// TIA Portal project "babu_washingMachineHMI" (V15)

(* hardware
DEVICE "S7-1200 station_1"  S7-1200 Station
   slot 0: "Rack_0"  S7-1200 Rack  Rack  V1.0
   slot 1: "PLC_1"  CPU 1212C DC/DC/DC  6ES7 212-1AE40-0XB0  V4.2
DEVICE "HMI_1"  KTP400 Basic PN
   slot 0: "HMI_1"  KTP400 Basic PN  6AV2 123-2DB03-0AX0  15.0.0.0
   slot 1: "HMI_RT_1"  KTP400 Basic PN  6AV2 123-2DB03-0AX0  15.0.0.0
   slot 5: "HMI_1.IE_CP_1"  PROFINET Interface  15.0.0.0
      slot 1: "PROFINET Interface_1"  PROFINET Interface
         slot 1: "Port_1"  Port
*)

// ===== PLC "PLC_1"  CPU 1212C DC/DC/DC =====

VAR_GLOBAL   // PLC tag table "Default tag table"
   "PUSH BUTTON ON" AT %M0.0 : Bool;
   "PUSH BUTTON ON MEM" AT %M0.1 : Bool;
   "PUSH BUTTON STOP" AT %M0.2 : Bool;
   "PUSH BUTTON STOP MEM" AT %M0.3 : Bool;
   "WATER AVAILABLE" AT %M0.4 : Bool;
   "WATER AVAILABLE MEM" AT %M0.5 : Bool;
   "DOOR CLOSED" AT %M0.6 : Bool;
   "DOOR CLOSED MEM" AT %M0.7 : Bool;
   "CLOTHS AVAILABLE MEM" AT %M1.0 : Bool;
   "CLOTHS AVAILABLE" AT %M1.1 : Bool;
   "CLEANING SOLUTION AVAILABLE" AT %M1.2 : Bool;
   "CLEANING SOLUTION AVAILABLE MEM" AT %M1.3 : Bool;
   "ALL OK TO START" AT %M1.4 : Bool;
   "OPEN SOLUTION INLET" AT %Q0.0 : Bool;
   "MOTOR CLOCKWISE" AT %Q0.1 : Bool;
   "MOTOR ANTI CLOCKWISE" AT %Q0.2 : Bool;
   "OPEN WATER OUTLET" AT %Q0.3 : Bool;
   "COMPLETED ALARM" AT %Q0.4 : Bool;
END_VAR

// folder: System blocks/Program resources

DATA_BLOCK "IEC_Timer_0_DB"   // DB1
{ S7_Optimized_Access := 'TRUE' }
AUTHOR : Simatic
FAMILY : IEC
NAME : IEC_TMR
VERSION : 1.0
// stored: InstanceOfName IEC_TIMER
"IEC_TIMER"
BEGIN
END_DATA_BLOCK

DATA_BLOCK "IEC_Timer_0_DB_1"   // DB2
{ S7_Optimized_Access := 'TRUE' }
AUTHOR : Simatic
FAMILY : IEC
NAME : IEC_TMR
VERSION : 1.0
// stored: InstanceOfName IEC_TIMER
"IEC_TIMER"
BEGIN
END_DATA_BLOCK

DATA_BLOCK "IEC_Timer_0_DB_2"   // DB3
{ S7_Optimized_Access := 'TRUE' }
AUTHOR : Simatic
FAMILY : IEC
NAME : IEC_TMR
VERSION : 1.0
// stored: InstanceOfName IEC_TIMER
"IEC_TIMER"
BEGIN
END_DATA_BLOCK

DATA_BLOCK "IEC_Timer_0_DB_3"   // DB4
{ S7_Optimized_Access := 'TRUE' }
AUTHOR : Simatic
FAMILY : IEC
NAME : IEC_TMR
VERSION : 1.0
// stored: InstanceOfName IEC_TIMER
"IEC_TIMER"
BEGIN
END_DATA_BLOCK

DATA_BLOCK "IEC_Timer_0_DB_4"   // DB5
{ S7_Optimized_Access := 'TRUE' }
AUTHOR : Simatic
FAMILY : IEC
NAME : IEC_TMR
VERSION : 1.0
// stored: InstanceOfName IEC_TIMER
"IEC_TIMER"
BEGIN
END_DATA_BLOCK

DATA_BLOCK "IEC_Timer_0_DB_5"   // DB6
{ S7_Optimized_Access := 'TRUE' }
AUTHOR : Simatic
FAMILY : IEC
NAME : IEC_TMR
VERSION : 1.0
// stored: InstanceOfName IEC_TIMER
"IEC_TIMER"
BEGIN
END_DATA_BLOCK

DATA_BLOCK "IEC_Timer_0_DB_6"   // DB7
{ S7_Optimized_Access := 'TRUE' }
AUTHOR : Simatic
FAMILY : IEC
NAME : IEC_TMR
VERSION : 1.0
// stored: InstanceOfName IEC_TIMER
"IEC_TIMER"
BEGIN
END_DATA_BLOCK

DATA_BLOCK "IEC_Timer_0_DB_7"   // DB8
{ S7_Optimized_Access := 'TRUE' }
AUTHOR : Simatic
FAMILY : IEC
NAME : IEC_TMR
VERSION : 1.0
// stored: InstanceOfName IEC_TIMER
"IEC_TIMER"
BEGIN
END_DATA_BLOCK

DATA_BLOCK "IEC_Timer_0_DB_8"   // DB9
{ S7_Optimized_Access := 'TRUE' }
AUTHOR : Simatic
FAMILY : IEC
NAME : IEC_TMR
VERSION : 1.0
// stored: InstanceOfName IEC_TIMER
"IEC_TIMER"
BEGIN
END_DATA_BLOCK

DATA_BLOCK "IEC_Timer_0_DB_9"   // DB10
{ S7_Optimized_Access := 'TRUE' }
AUTHOR : Simatic
FAMILY : IEC
NAME : IEC_TMR
VERSION : 1.0
// stored: InstanceOfName IEC_TIMER
"IEC_TIMER"
BEGIN
END_DATA_BLOCK

DATA_BLOCK "IEC_Timer_0_DB_10"   // DB11
{ S7_Optimized_Access := 'TRUE' }
AUTHOR : Simatic
FAMILY : IEC
NAME : IEC_TMR
VERSION : 1.0
// stored: InstanceOfName IEC_TIMER
"IEC_TIMER"
BEGIN
END_DATA_BLOCK

DATA_BLOCK "IEC_Timer_0_DB_11"   // DB12
{ S7_Optimized_Access := 'TRUE' }
AUTHOR : Simatic
FAMILY : IEC
NAME : IEC_TMR
VERSION : 1.0
// stored: InstanceOfName IEC_TIMER
"IEC_TIMER"
BEGIN
END_DATA_BLOCK

DATA_BLOCK "IEC_Timer_0_DB_12"   // DB13
{ S7_Optimized_Access := 'TRUE' }
AUTHOR : Simatic
FAMILY : IEC
NAME : IEC_TMR
VERSION : 1.0
// stored: InstanceOfName IEC_TIMER
"IEC_TIMER"
BEGIN
END_DATA_BLOCK

DATA_BLOCK "IEC_Timer_0_DB_13"   // DB14
{ S7_Optimized_Access := 'TRUE' }
AUTHOR : Simatic
FAMILY : IEC
NAME : IEC_TMR
VERSION : 1.0
// stored: InstanceOfName IEC_TIMER
"IEC_TIMER"
BEGIN
END_DATA_BLOCK

// folder: (top level)

ORGANIZATION_BLOCK "Main"   // OB1, LAD, ProgramCycle
TITLE = "Main Program Sweep (Cycle)"
{ S7_Optimized_Access := 'TRUE' }
VERSION : 0.1
   VAR_INPUT
      Initial_Call : Bool;   // Initial call of this OB
      Remanence : Bool;   // =True, if remanent data are available
   END_VAR
BEGIN

REGION Network 1
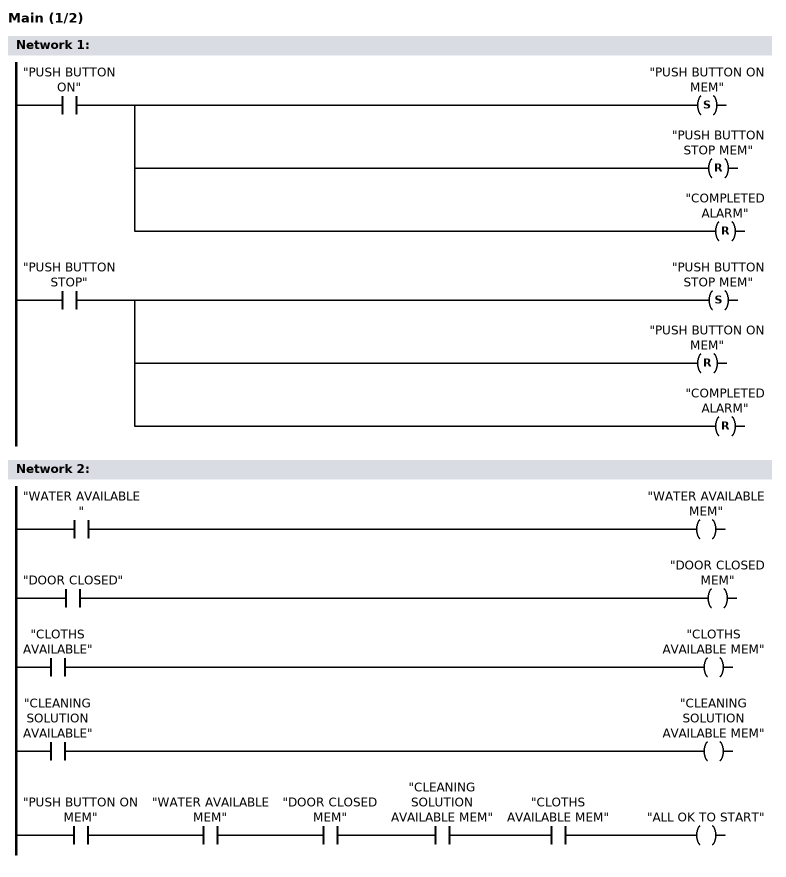
   RUNG wire#powerrail
      Contact( "PUSH BUTTON ON" )
      wire#w1
      S_Coil( "PUSH BUTTON ON MEM" )
   END_RUNG
   RUNG wire#w1
      R_Coil( "PUSH BUTTON STOP MEM" )
   END_RUNG
   RUNG wire#w1
      R_Coil( "COMPLETED ALARM" )
   END_RUNG
   RUNG wire#powerrail
      Contact( "PUSH BUTTON STOP" )
      wire#w2
      S_Coil( "PUSH BUTTON STOP MEM" )
   END_RUNG
   RUNG wire#w2
      R_Coil( "PUSH BUTTON ON MEM" )
   END_RUNG
   RUNG wire#w2
      R_Coil( "COMPLETED ALARM" )
   END_RUNG
   // the same network as SCL:
   IF "PUSH BUTTON ON" THEN
       "PUSH BUTTON ON MEM" := TRUE;
       "PUSH BUTTON STOP MEM" := FALSE;
       "COMPLETED ALARM" := FALSE;
   END_IF;
   IF "PUSH BUTTON STOP" THEN
       "PUSH BUTTON STOP MEM" := TRUE;
       "PUSH BUTTON ON MEM" := FALSE;
       "COMPLETED ALARM" := FALSE;
   END_IF;
END_REGION

REGION Network 2
   RUNG wire#powerrail
      Contact( "WATER AVAILABLE" )
      Coil( "WATER AVAILABLE MEM" )
   END_RUNG
   RUNG wire#powerrail
      Contact( "DOOR CLOSED" )
      Coil( "DOOR CLOSED MEM" )
   END_RUNG
   RUNG wire#powerrail
      Contact( "CLOTHS AVAILABLE" )
      Coil( "CLOTHS AVAILABLE MEM" )
   END_RUNG
   RUNG wire#powerrail
      Contact( "CLEANING SOLUTION AVAILABLE" )
      Coil( "CLEANING SOLUTION AVAILABLE MEM" )
   END_RUNG
   RUNG wire#powerrail
      Contact( "PUSH BUTTON ON MEM" )
      Contact( "WATER AVAILABLE MEM" )
      Contact( "DOOR CLOSED MEM" )
      Contact( "CLEANING SOLUTION AVAILABLE MEM" )
      Contact( "CLOTHS AVAILABLE MEM" )
      Coil( "ALL OK TO START" )
   END_RUNG
   // the same network as SCL:
   "WATER AVAILABLE MEM" := "WATER AVAILABLE";
   "DOOR CLOSED MEM" := "DOOR CLOSED";
   "CLOTHS AVAILABLE MEM" := "CLOTHS AVAILABLE";
   "CLEANING SOLUTION AVAILABLE MEM" := "CLEANING SOLUTION AVAILABLE";
   "ALL OK TO START" := "PUSH BUTTON ON MEM" AND "WATER AVAILABLE MEM" AND "DOOR CLOSED MEM" AND "CLEANING SOLUTION AVAILABLE MEM" AND "CLOTHS AVAILABLE MEM";
END_REGION

REGION Network 3
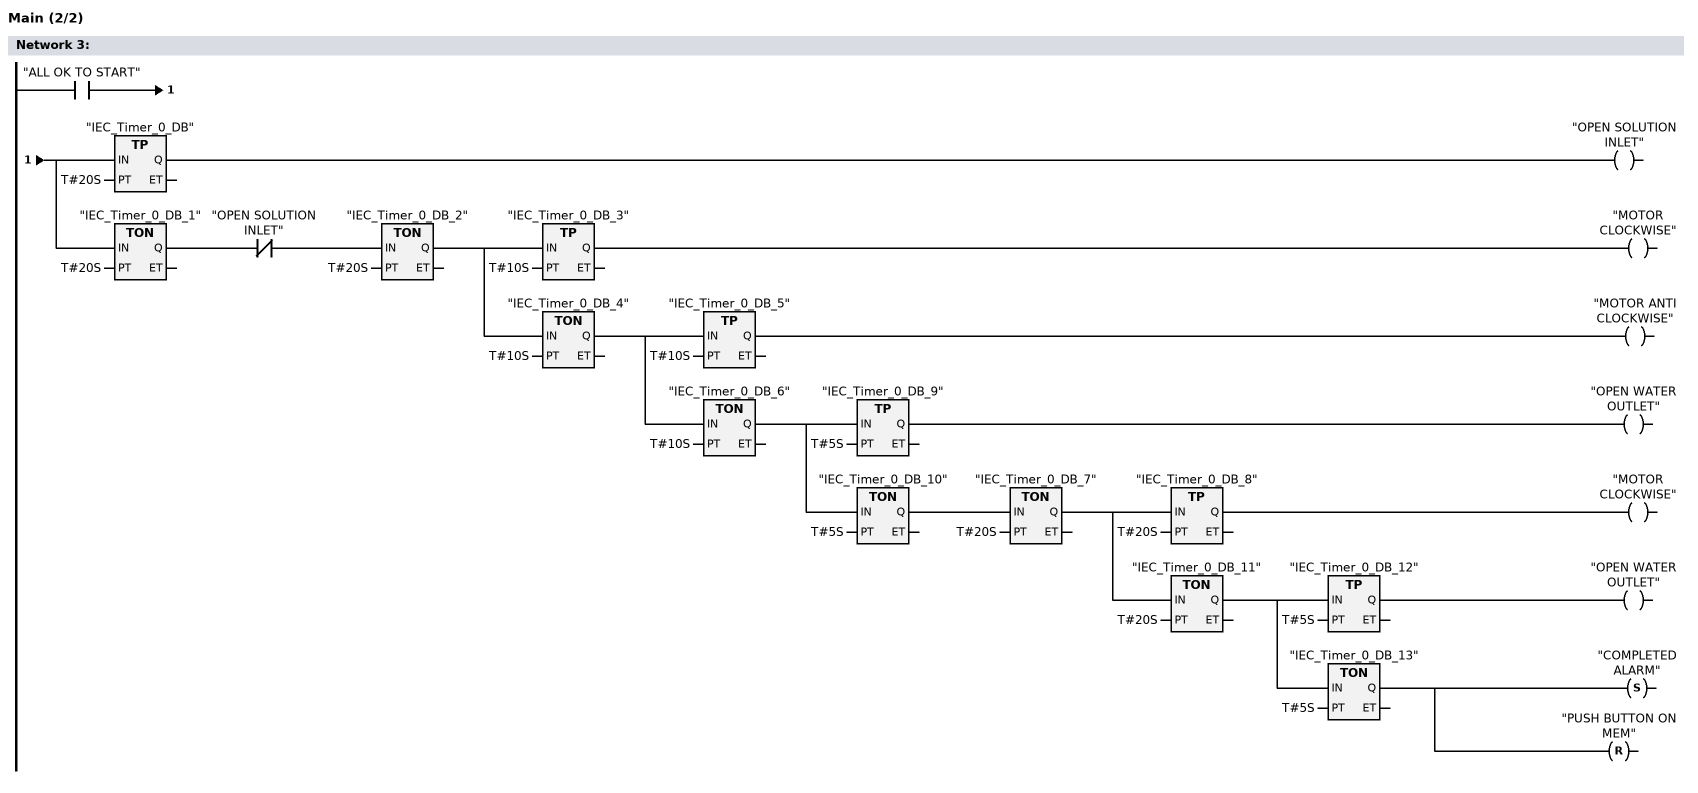
   "IEC_Timer_0_DB".TP(IN := "ALL OK TO START", PT := T#20S);
   "OPEN SOLUTION INLET" := "IEC_Timer_0_DB".Q;
   "IEC_Timer_0_DB_1".TON(IN := "ALL OK TO START", PT := T#20S);
   "IEC_Timer_0_DB_2".TON(IN := "IEC_Timer_0_DB_1".Q AND NOT "OPEN SOLUTION INLET", PT := T#20S);
   "IEC_Timer_0_DB_3".TP(IN := "IEC_Timer_0_DB_2".Q, PT := T#10S);
   "MOTOR CLOCKWISE" := "IEC_Timer_0_DB_3".Q;
   "IEC_Timer_0_DB_4".TON(IN := "IEC_Timer_0_DB_2".Q, PT := T#10S);
   "IEC_Timer_0_DB_5".TP(IN := "IEC_Timer_0_DB_4".Q, PT := T#10S);
   "MOTOR ANTI CLOCKWISE" := "IEC_Timer_0_DB_5".Q;
   "IEC_Timer_0_DB_6".TON(IN := "IEC_Timer_0_DB_4".Q, PT := T#10S);
   "IEC_Timer_0_DB_9".TP(IN := "IEC_Timer_0_DB_6".Q, PT := T#5S);
   "OPEN WATER OUTLET" := "IEC_Timer_0_DB_9".Q;
   "IEC_Timer_0_DB_10".TON(IN := "IEC_Timer_0_DB_6".Q, PT := T#5S);
   "IEC_Timer_0_DB_7".TON(IN := "IEC_Timer_0_DB_10".Q, PT := T#20S);
   "IEC_Timer_0_DB_8".TP(IN := "IEC_Timer_0_DB_7".Q, PT := T#20S);
   "MOTOR CLOCKWISE" := "IEC_Timer_0_DB_8".Q;
   "IEC_Timer_0_DB_11".TON(IN := "IEC_Timer_0_DB_7".Q, PT := T#20S);
   "IEC_Timer_0_DB_12".TP(IN := "IEC_Timer_0_DB_11".Q, PT := T#5S);
   "OPEN WATER OUTLET" := "IEC_Timer_0_DB_12".Q;
   "IEC_Timer_0_DB_13".TON(IN := "IEC_Timer_0_DB_11".Q, PT := T#5S);
   IF "IEC_Timer_0_DB_13".Q THEN
       "COMPLETED ALARM" := TRUE;
       "PUSH BUTTON ON MEM" := FALSE;
   END_IF;
END_REGION
END_ORGANIZATION_BLOCK

(* ===== HMI "HMI_RT_1" =====
connection "HMI_Connection_1": ETHERNET, SMART_S7_1200_OMS

screen "Root screen" 480x272, template "Template_1"
   Switch "Pushbutton_Round_G" at 9,9 size 50x50; CaptionText 'Switch'; TextOff '0'; TextOn '1'; PictureOff "Pushbutton_Round_G_Off_256c"; PictureOn "Pushbutton_Round_G_On_256c"
   Switch "Pushbutton_Round_R" at 9,67 size 50x50; CaptionText 'Switch'; TextOff '0'; TextOn '1'; PictureOff "Pushbutton_Round_R_Off_256c"; PictureOn "Pushbutton_Round_R_On_256c"
*)